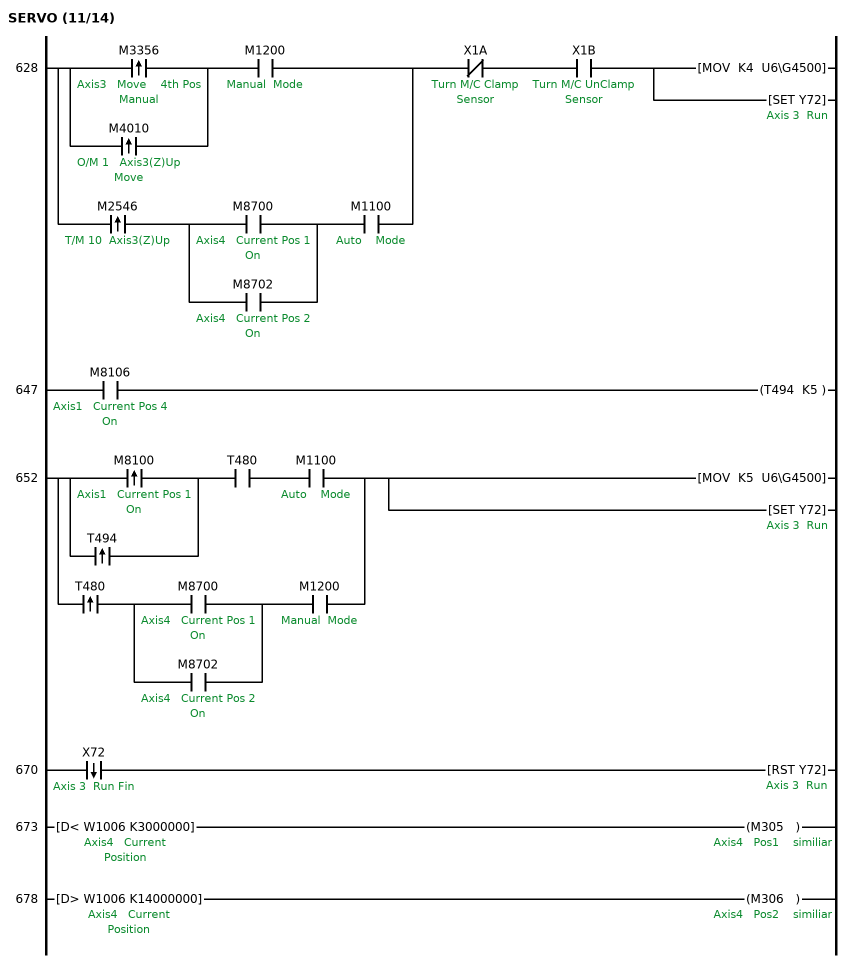
[picture p48: ladder of SERVO, rungs at steps 628 to 678]
628   LDP     M3356  ; Axis3   Move    4th Pos Manual
      ORP     M4010  ; O/M 1   Axis3(Z)Up Move
      AND     M1200  ; Manual  Mode
      LDP     M2546  ; T/M 10  Axis3(Z)Up
      LD      M8700  ; Axis4   Current Pos 1 On
      OR      M8702  ; Axis4   Current Pos 2 On
      ANB
      AND     M1100  ; Auto    Mode
      ORB
      ANI     X1A  ; Turn M/C Clamp Sensor
      AND     X1B  ; Turn M/C UnClamp Sensor
      MOV     K4 U6\G4500
      SET     Y72  ; Axis 3  Run
647   LD      M8106  ; Axis1   Current Pos 4 On
      OUT     T494 K5
652   LDP     M8100  ; Axis1   Current Pos 1 On
      ORP     T494
      AND     T480
      AND     M1100  ; Auto    Mode
      LDP     T480
      LD      M8700  ; Axis4   Current Pos 1 On
      OR      M8702  ; Axis4   Current Pos 2 On
      ANB
      AND     M1200  ; Manual  Mode
      ORB
      MOV     K5 U6\G4500
      SET     Y72  ; Axis 3  Run
670   LDF     X72  ; Axis 3  Run Fin
      RST     Y72  ; Axis 3  Run
673   LDD<    W1006 K3000000  ; Axis4   Current Position
      OUT     M305  ; Axis4   Pos1    similiar
678   LDD>    W1006 K14000000  ; Axis4   Current Position
      OUT     M306  ; Axis4   Pos2    similiar
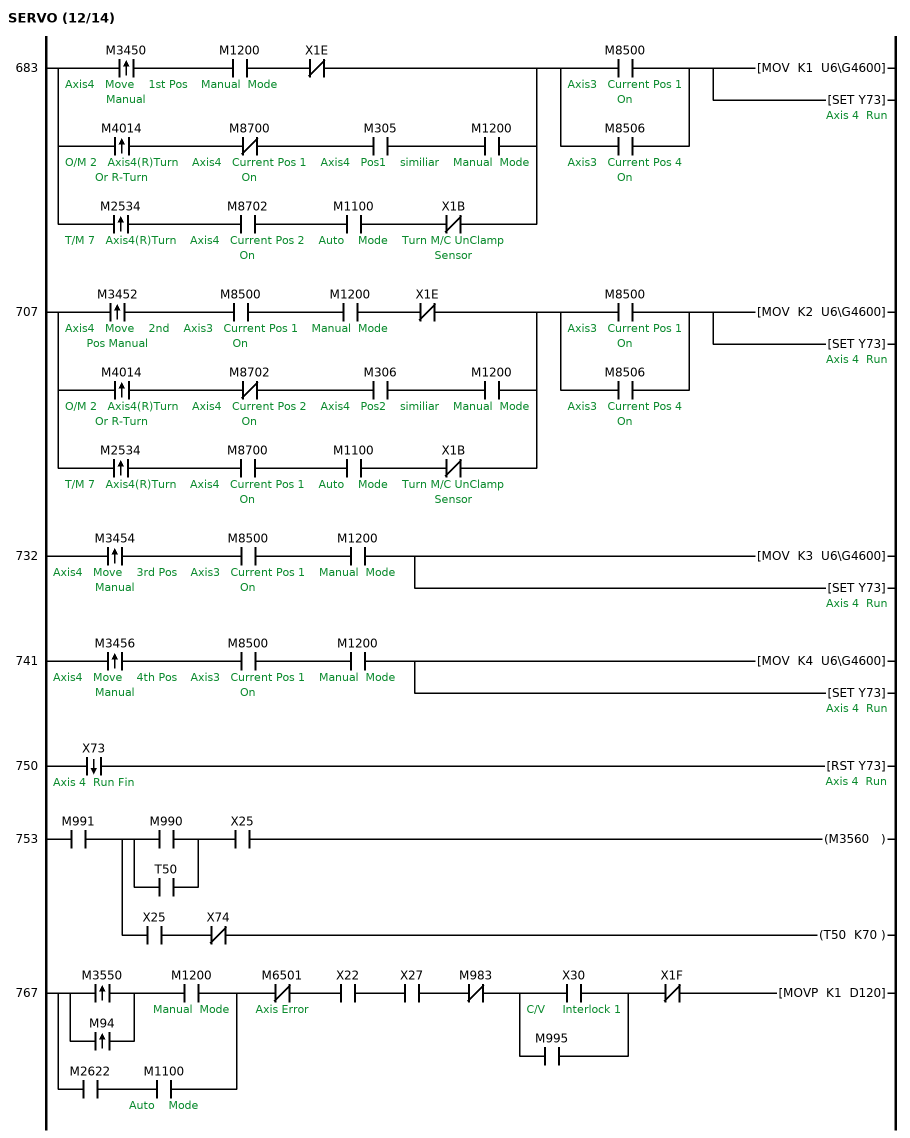
683   LDP     M3450  ; Axis4   Move    1st Pos Manual
      AND     M1200  ; Manual  Mode
      ANI     X1E
      LDP     M4014  ; O/M 2   Axis4(R)Turn Or R-Turn
      ANI     M8700  ; Axis4   Current Pos 1 On
      AND     M305  ; Axis4   Pos1    similiar
      AND     M1200  ; Manual  Mode
      ORB
      LDP     M2534  ; T/M 7   Axis4(R)Turn
      AND     M8702  ; Axis4   Current Pos 2 On
      AND     M1100  ; Auto    Mode
      ANI     X1B  ; Turn M/C UnClamp Sensor
      ORB
      LD      M8500  ; Axis3   Current Pos 1 On
      OR      M8506  ; Axis3   Current Pos 4 On
      ANB
      MOV     K1 U6\G4600
      SET     Y73  ; Axis 4  Run
707   LDP     M3452  ; Axis4   Move    2nd Pos Manual
      AND     M8500  ; Axis3   Current Pos 1 On
      AND     M1200  ; Manual  Mode
      ANI     X1E
      LDP     M4014  ; O/M 2   Axis4(R)Turn Or R-Turn
      ANI     M8702  ; Axis4   Current Pos 2 On
      AND     M306  ; Axis4   Pos2    similiar
      AND     M1200  ; Manual  Mode
      ORB
      LDP     M2534  ; T/M 7   Axis4(R)Turn
      AND     M8700  ; Axis4   Current Pos 1 On
      AND     M1100  ; Auto    Mode
      ANI     X1B  ; Turn M/C UnClamp Sensor
      ORB
      LD      M8500  ; Axis3   Current Pos 1 On
      OR      M8506  ; Axis3   Current Pos 4 On
      ANB
      MOV     K2 U6\G4600
      SET     Y73  ; Axis 4  Run
732   LDP     M3454  ; Axis4   Move    3rd Pos Manual
      AND     M8500  ; Axis3   Current Pos 1 On
      AND     M1200  ; Manual  Mode
      MOV     K3 U6\G4600
      SET     Y73  ; Axis 4  Run
741   LDP     M3456  ; Axis4   Move    4th Pos Manual
      AND     M8500  ; Axis3   Current Pos 1 On
      AND     M1200  ; Manual  Mode
      MOV     K4 U6\G4600
      SET     Y73  ; Axis 4  Run
750   LDF     X73  ; Axis 4  Run Fin
      RST     Y73  ; Axis 4  Run
753   LD      M991
      MPS
      LD      M990
      OR      T50
      ANB
      AND     X25
      OUT     M3560
      MPP
      AND     X25
      ANI     X74
      OUT     T50 K70
767   LDP     M3550
      ORP     M94
      AND     M1200  ; Manual  Mode
      LD      M2622
      AND     M1100  ; Auto    Mode
      ORB
      ANI     M6501  ; Axis Error
      AND     X22
      AND     X27
      ANI     M983
      LD      X30  ; C/V     Interlock 1
      OR      M995
      ANB
      ANI     X1F
      MOVP    K1 D120
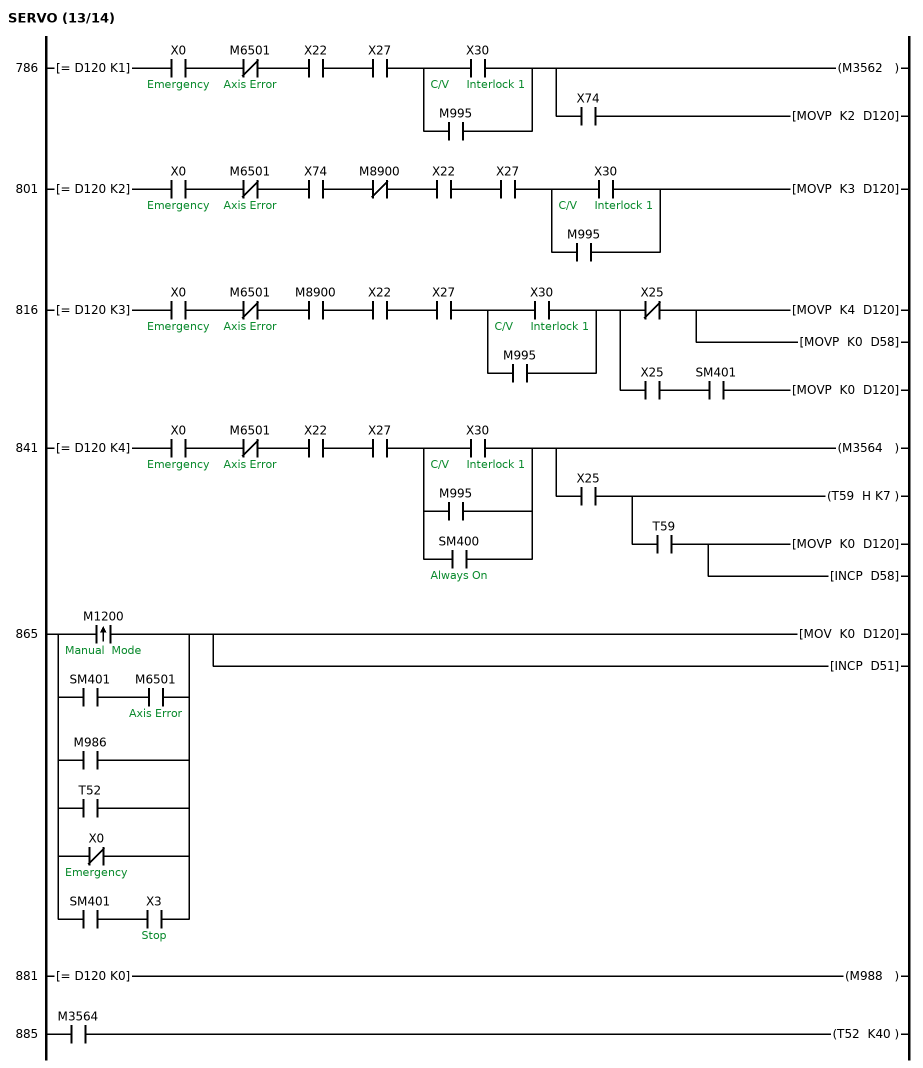
786   LD=     D120 K1
      AND     X0  ; Emergency
      ANI     M6501  ; Axis Error
      AND     X22
      AND     X27
      LD      X30  ; C/V     Interlock 1
      OR      M995
      ANB
      OUT     M3562
      AND     X74
      MOVP    K2 D120
801   LD=     D120 K2
      AND     X0  ; Emergency
      ANI     M6501  ; Axis Error
      AND     X74
      ANI     M8900
      AND     X22
      AND     X27
      LD      X30  ; C/V     Interlock 1
      OR      M995
      ANB
      MOVP    K3 D120
816   LD=     D120 K3
      AND     X0  ; Emergency
      ANI     M6501  ; Axis Error
      AND     M8900
      AND     X22
      AND     X27
      LD      X30  ; C/V     Interlock 1
      OR      M995
      ANB
      MPS
      ANI     X25
      MOVP    K4 D120
      MOVP    K0 D58
      MPP
      AND     X25
      AND     SM401
      MOVP    K0 D120
841   LD=     D120 K4
      AND     X0  ; Emergency
      ANI     M6501  ; Axis Error
      AND     X22
      AND     X27
      LD      X30  ; C/V     Interlock 1
      OR      M995
      OR      SM400  ; Always On
      ANB
      OUT     M3564
      AND     X25
      OUTH    T59 K7
      AND     T59
      MOVP    K0 D120
      INCP    D58
865   LDP     M1200  ; Manual  Mode
      LD      SM401
      AND     M6501  ; Axis Error
      ORB
      OR      M986
      OR      T52
      ORI     X0  ; Emergency
      LD      SM401
      AND     X3  ; Stop
      ORB
      MOV     K0 D120
      INCP    D51
881   LD=     D120 K0
      OUT     M988
885   LD      M3564
      OUT     T52 K40
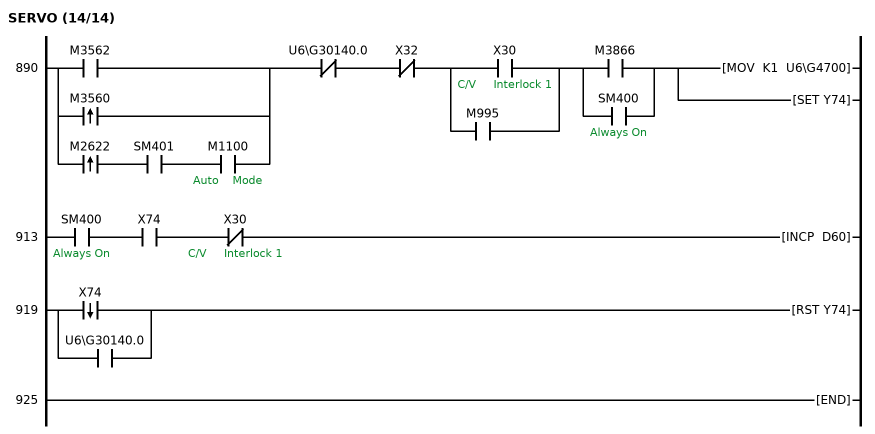
890   LD      M3562
      ORP     M3560
      LDP     M2622
      AND     SM401
      AND     M1100  ; Auto    Mode
      ORB
      ANI     U6\G30140.0
      ANI     X32
      LD      X30  ; C/V     Interlock 1
      OR      M995
      ANB
      LD      M3866
      OR      SM400  ; Always On
      ANB
      MOV     K1 U6\G4700
      SET     Y74
913   LD      SM400  ; Always On
      AND     X74
      ANI     X30  ; C/V     Interlock 1
      INCP    D60
919   LDF     X74
      OR      U6\G30140.0
      RST     Y74
925   END
END_PROGRAM

PROGRAM Y_OUT
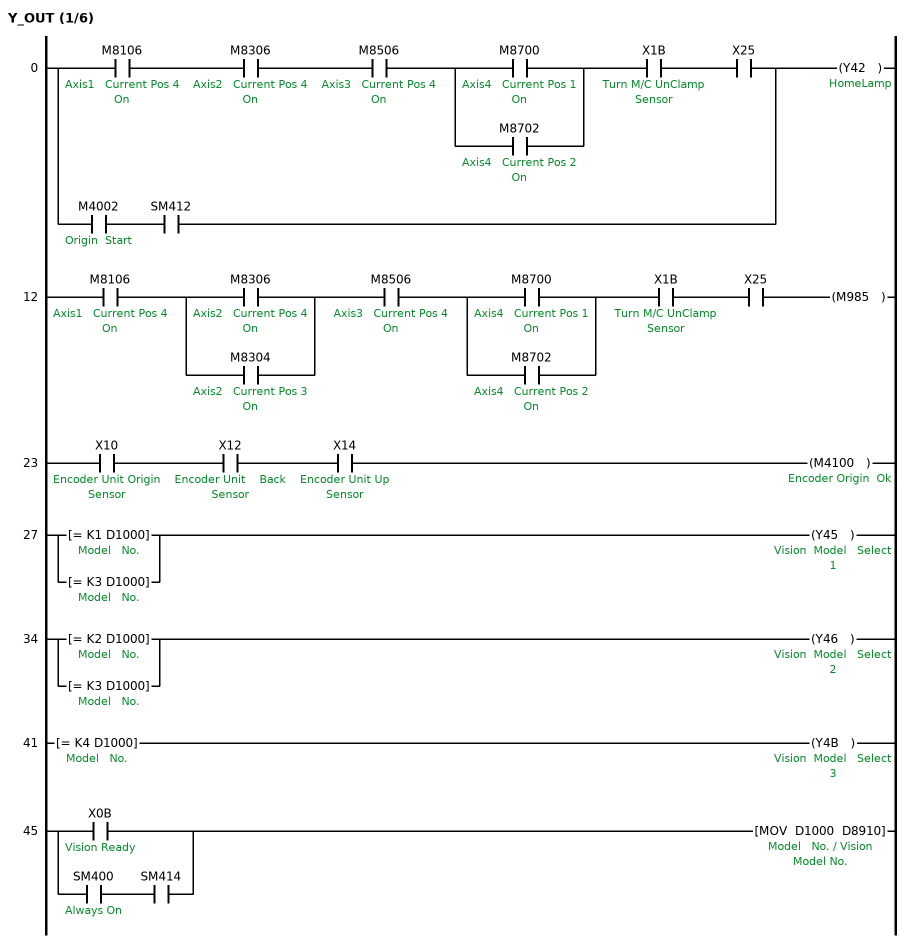
0     LD      M8106  ; Axis1   Current Pos 4 On
      AND     M8306  ; Axis2   Current Pos 4 On
      AND     M8506  ; Axis3   Current Pos 4 On
      LD      M8700  ; Axis4   Current Pos 1 On
      OR      M8702  ; Axis4   Current Pos 2 On
      ANB
      AND     X1B  ; Turn M/C UnClamp Sensor
      AND     X25
      LD      M4002  ; Origin  Start
      AND     SM412
      ORB
      OUT     Y42  ; HomeLamp
12    LD      M8106  ; Axis1   Current Pos 4 On
      LD      M8306  ; Axis2   Current Pos 4 On
      OR      M8304  ; Axis2   Current Pos 3 On
      ANB
      AND     M8506  ; Axis3   Current Pos 4 On
      LD      M8700  ; Axis4   Current Pos 1 On
      OR      M8702  ; Axis4   Current Pos 2 On
      ANB
      AND     X1B  ; Turn M/C UnClamp Sensor
      AND     X25
      OUT     M985
23    LD      X10  ; Encoder Unit Origin Sensor
      AND     X12  ; Encoder Unit    Back    Sensor
      AND     X14  ; Encoder Unit Up Sensor
      OUT     M4100  ; Encoder Origin  Ok
27    LD=     K1 D1000  ; Model   No.
      OR=     K3 D1000  ; Model   No.
      OUT     Y45  ; Vision  Model   Select 1
34    LD=     K2 D1000  ; Model   No.
      OR=     K3 D1000  ; Model   No.
      OUT     Y46  ; Vision  Model   Select 2
41    LD=     K4 D1000  ; Model   No.
      OUT     Y4B  ; Vision  Model   Select 3
45    LD      X0B  ; Vision Ready
      LD      SM400  ; Always On
      AND     SM414
      ORB
      MOV     D1000 D8910  ; Vision Model No.
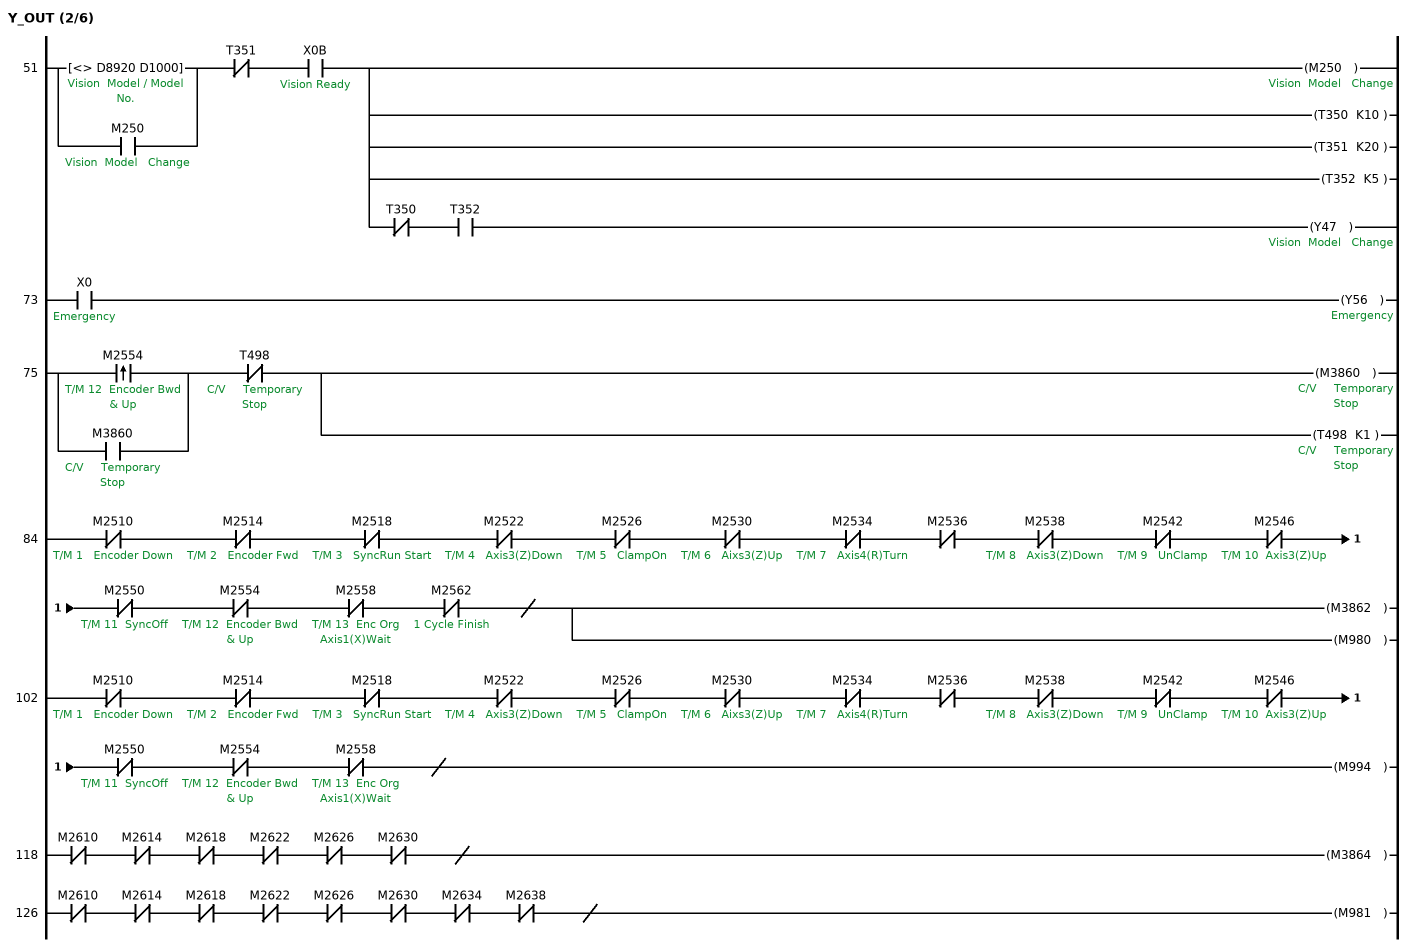
51    LD<>    D8920 D1000  ; Vision  Model / Model   No.
      OR      M250  ; Vision  Model   Change
      ANI     T351
      AND     X0B  ; Vision Ready
      OUT     M250  ; Vision  Model   Change
      OUT     T350 K10
      OUT     T351 K20
      OUT     T352 K5
      ANI     T350
      AND     T352
      OUT     Y47  ; Vision  Model   Change
73    LD      X0  ; Emergency
      OUT     Y56  ; Emergency
75    LDP     M2554  ; T/M 12  Encoder Bwd & Up
      OR      M3860  ; C/V     Temporary  Stop
      ANI     T498  ; C/V     Temporary  Stop
      OUT     M3860  ; C/V     Temporary  Stop
      OUT     T498 K1  ; C/V     Temporary  Stop
84    LDI     M2510  ; T/M 1   Encoder Down
      ANI     M2514  ; T/M 2   Encoder Fwd
      ANI     M2518  ; T/M 3   SyncRun Start
      ANI     M2522  ; T/M 4   Axis3(Z)Down
      ANI     M2526  ; T/M 5   ClampOn
      ANI     M2530  ; T/M 6   Aixs3(Z)Up
      ANI     M2534  ; T/M 7   Axis4(R)Turn
      ANI     M2536
      ANI     M2538  ; T/M 8   Axis3(Z)Down
      ANI     M2542  ; T/M 9   UnClamp
      ANI     M2546  ; T/M 10  Axis3(Z)Up
      ANI     M2550  ; T/M 11  SyncOff
      ANI     M2554  ; T/M 12  Encoder Bwd & Up
      ANI     M2558  ; T/M 13  Enc Org Axis1(X)Wait
      ANI     M2562  ; 1 Cycle Finish
      INV
      OUT     M3862
      OUT     M980
102   LDI     M2510  ; T/M 1   Encoder Down
      ANI     M2514  ; T/M 2   Encoder Fwd
      ANI     M2518  ; T/M 3   SyncRun Start
      ANI     M2522  ; T/M 4   Axis3(Z)Down
      ANI     M2526  ; T/M 5   ClampOn
      ANI     M2530  ; T/M 6   Aixs3(Z)Up
      ANI     M2534  ; T/M 7   Axis4(R)Turn
      ANI     M2536
      ANI     M2538  ; T/M 8   Axis3(Z)Down
      ANI     M2542  ; T/M 9   UnClamp
      ANI     M2546  ; T/M 10  Axis3(Z)Up
      ANI     M2550  ; T/M 11  SyncOff
      ANI     M2554  ; T/M 12  Encoder Bwd & Up
      ANI     M2558  ; T/M 13  Enc Org Axis1(X)Wait
      INV
      OUT     M994
118   LDI     M2610
      ANI     M2614
      ANI     M2618
      ANI     M2622
      ANI     M2626
      ANI     M2630
      INV
      OUT     M3864
126   LDI     M2610
      ANI     M2614
      ANI     M2618
      ANI     M2622
      ANI     M2626
      ANI     M2630
      ANI     M2634
      ANI     M2638
      INV
      OUT     M981
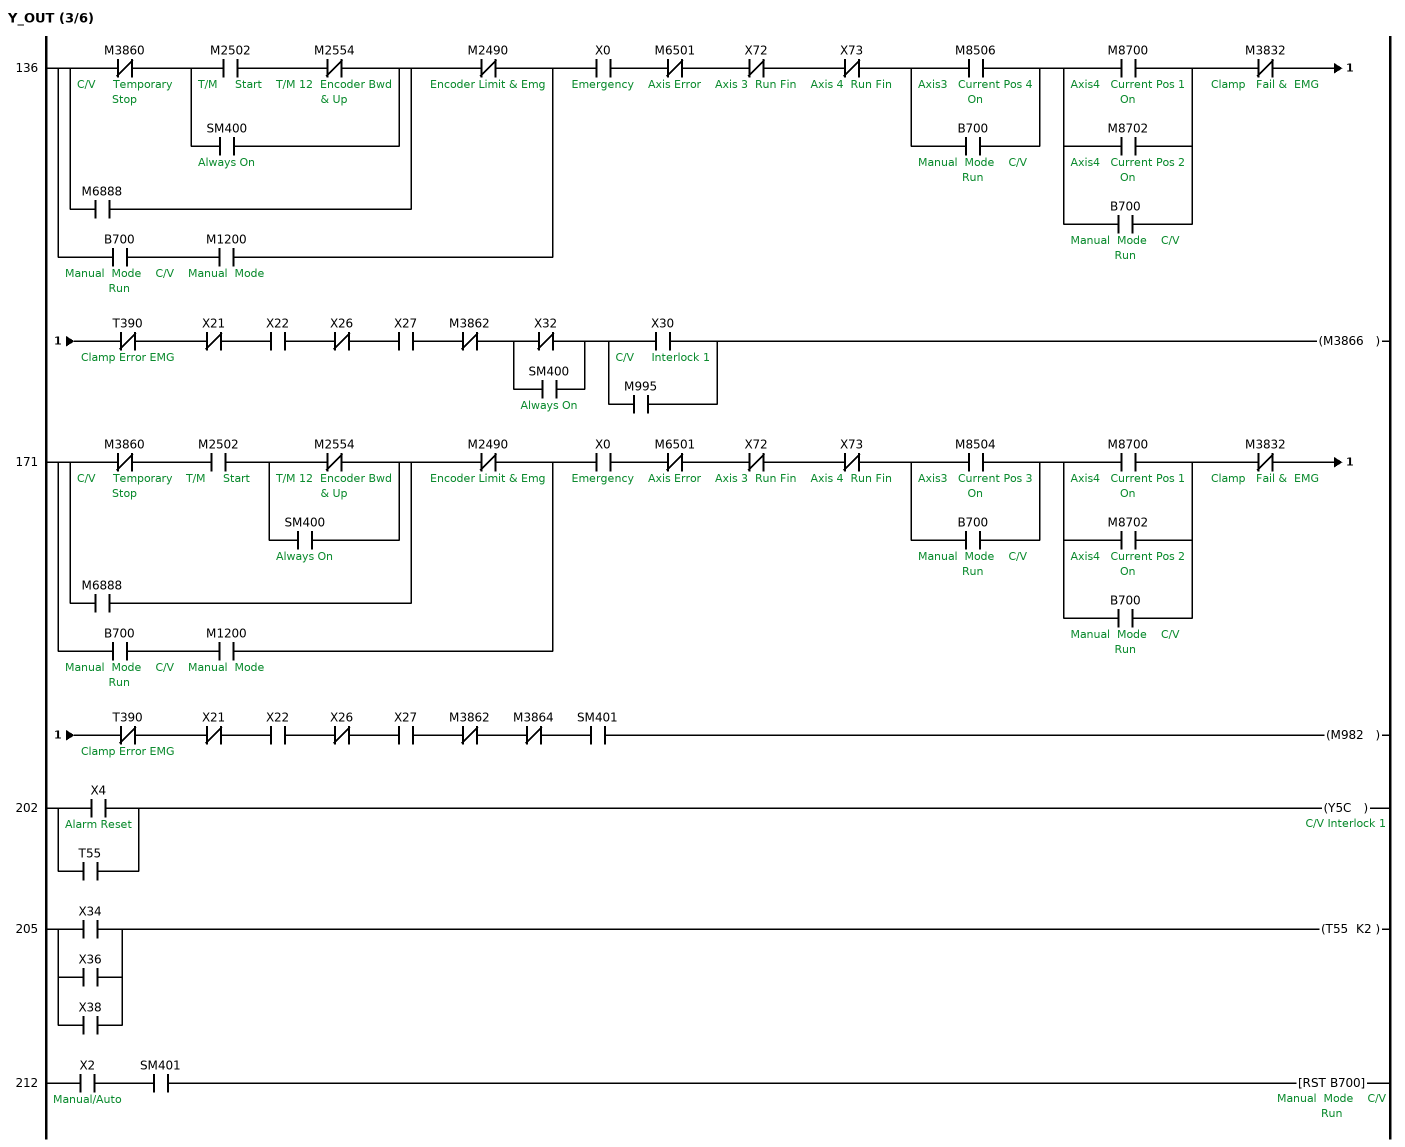
136   LDI     M3860  ; C/V     Temporary  Stop
      LD      M2502  ; T/M     Start
      ANI     M2554  ; T/M 12  Encoder Bwd & Up
      OR      SM400  ; Always On
      ANB
      OR      M6888
      ANI     M2490  ; Encoder Limit & Emg
      LD      B700  ; Manual  Mode    C/V Run
      AND     M1200  ; Manual  Mode
      ORB
      AND     X0  ; Emergency
      ANI     M6501  ; Axis Error
      ANI     X72  ; Axis 3  Run Fin
      ANI     X73  ; Axis 4  Run Fin
      LD      M8506  ; Axis3   Current Pos 4 On
      OR      B700  ; Manual  Mode    C/V Run
      ANB
      LD      M8700  ; Axis4   Current Pos 1 On
      OR      M8702  ; Axis4   Current Pos 2 On
      OR      B700  ; Manual  Mode    C/V Run
      ANB
      ANI     M3832  ; Clamp   Fail &  EMG
      ANI     T390  ; Clamp Error EMG
      ANI     X21
      AND     X22
      ANI     X26
      AND     X27
      ANI     M3862
      LDI     X32
      OR      SM400  ; Always On
      ANB
      LD      X30  ; C/V     Interlock 1
      OR      M995
      ANB
      OUT     M3866
171   LDI     M3860  ; C/V     Temporary  Stop
      AND     M2502  ; T/M     Start
      LDI     M2554  ; T/M 12  Encoder Bwd & Up
      OR      SM400  ; Always On
      ANB
      OR      M6888
      ANI     M2490  ; Encoder Limit & Emg
      LD      B700  ; Manual  Mode    C/V Run
      AND     M1200  ; Manual  Mode
      ORB
      AND     X0  ; Emergency
      ANI     M6501  ; Axis Error
      ANI     X72  ; Axis 3  Run Fin
      ANI     X73  ; Axis 4  Run Fin
      LD      M8504  ; Axis3   Current Pos 3 On
      OR      B700  ; Manual  Mode    C/V Run
      ANB
      LD      M8700  ; Axis4   Current Pos 1 On
      OR      M8702  ; Axis4   Current Pos 2 On
      OR      B700  ; Manual  Mode    C/V Run
      ANB
      ANI     M3832  ; Clamp   Fail &  EMG
      ANI     T390  ; Clamp Error EMG
      ANI     X21
      AND     X22
      ANI     X26
      AND     X27
      ANI     M3862
      ANI     M3864
      AND     SM401
      OUT     M982
202   LD      X4  ; Alarm Reset
      OR      T55
      OUT     Y5C  ; C/V Interlock 1
205   LD      X34
      OR      X36
      OR      X38
      OUT     T55 K2
212   LD      X2  ; Manual/Auto
      AND     SM401
      RST     B700  ; Manual  Mode    C/V Run
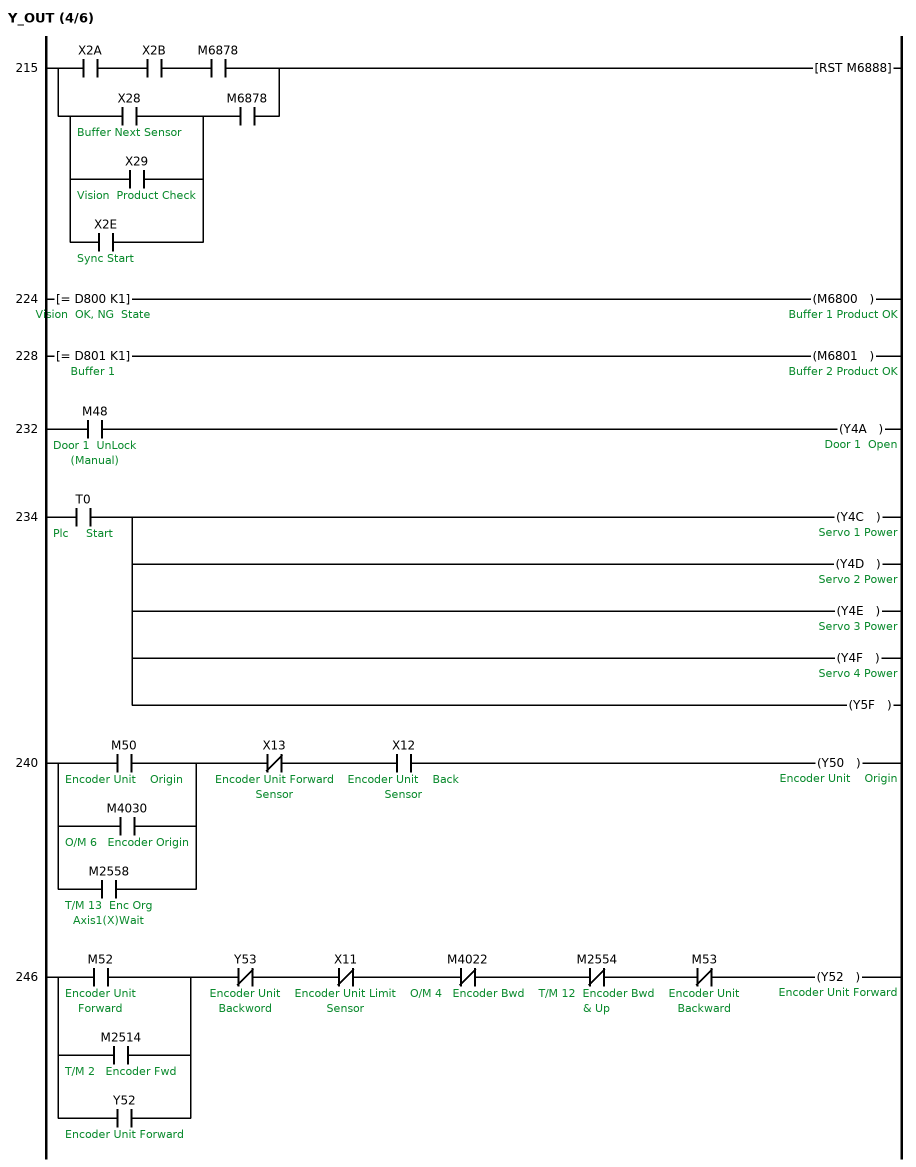
215   LD      X2A
      AND     X2B
      AND     M6878
      LD      X28  ; Buffer Next Sensor
      OR      X29  ; Vision  Product Check
      OR      X2E  ; Sync Start
      AND     M6878
      ORB
      RST     M6888
224   LD=     D800 K1  ; Vision  OK, NG  State
      OUT     M6800  ; Buffer 1 Product OK
228   LD=     D801 K1  ; Buffer 1
      OUT     M6801  ; Buffer 2 Product OK
232   LD      M48  ; Door 1  UnLock  (Manual)
      OUT     Y4A  ; Door 1  Open
234   LD      T0  ; Plc     Start
      OUT     Y4C  ; Servo 1 Power
      OUT     Y4D  ; Servo 2 Power
      OUT     Y4E  ; Servo 3 Power
      OUT     Y4F  ; Servo 4 Power
      OUT     Y5F
240   LD      M50  ; Encoder Unit    Origin
      OR      M4030  ; O/M 6   Encoder Origin
      OR      M2558  ; T/M 13  Enc Org Axis1(X)Wait
      ANI     X13  ; Encoder Unit Forward Sensor
      AND     X12  ; Encoder Unit    Back    Sensor
      OUT     Y50  ; Encoder Unit    Origin
246   LD      M52  ; Encoder Unit    Forward
      OR      M2514  ; T/M 2   Encoder Fwd
      OR      Y52  ; Encoder Unit Forward
      ANI     Y53  ; Encoder Unit Backword
      ANI     X11  ; Encoder Unit Limit Sensor
      ANI     M4022  ; O/M 4   Encoder Bwd
      ANI     M2554  ; T/M 12  Encoder Bwd & Up
      ANI     M53  ; Encoder Unit    Backward
      OUT     Y52  ; Encoder Unit Forward
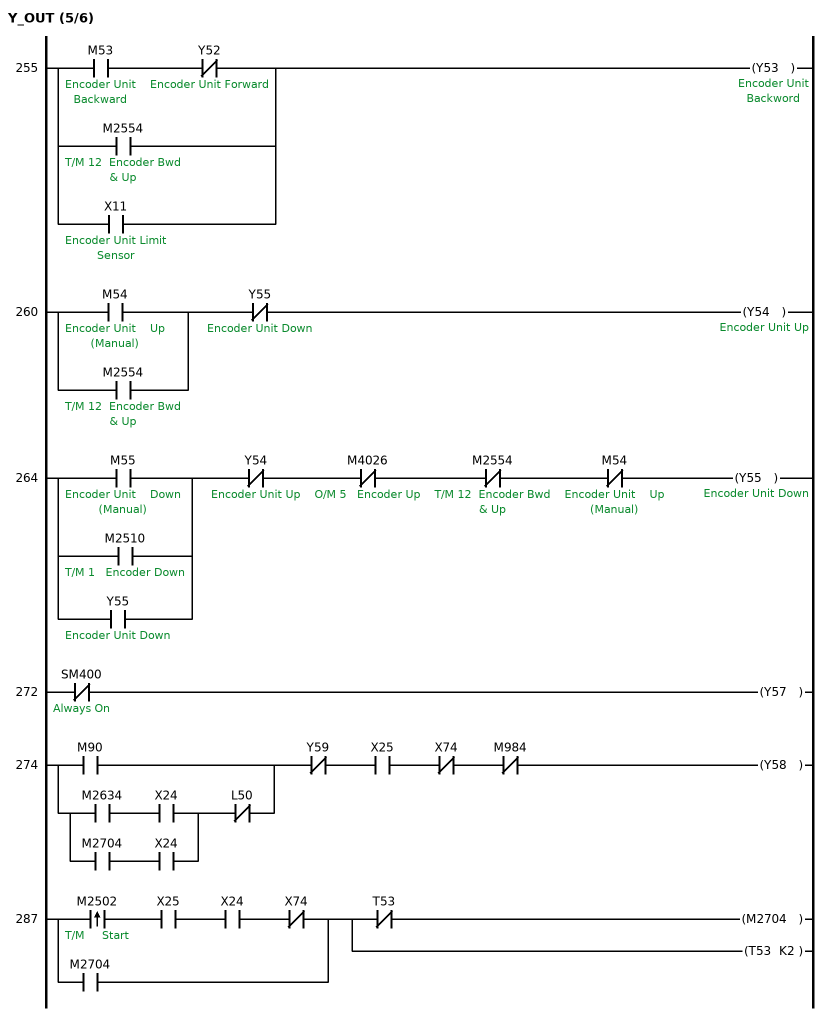
255   LD      M53  ; Encoder Unit    Backward
      ANI     Y52  ; Encoder Unit Forward
      OR      M2554  ; T/M 12  Encoder Bwd & Up
      OR      X11  ; Encoder Unit Limit Sensor
      OUT     Y53  ; Encoder Unit Backword
260   LD      M54  ; Encoder Unit    Up      (Manual)
      OR      M2554  ; T/M 12  Encoder Bwd & Up
      ANI     Y55  ; Encoder Unit Down
      OUT     Y54  ; Encoder Unit Up
264   LD      M55  ; Encoder Unit    Down    (Manual)
      OR      M2510  ; T/M 1   Encoder Down
      OR      Y55  ; Encoder Unit Down
      ANI     Y54  ; Encoder Unit Up
      ANI     M4026  ; O/M 5   Encoder Up
      ANI     M2554  ; T/M 12  Encoder Bwd & Up
      ANI     M54  ; Encoder Unit    Up      (Manual)
      OUT     Y55  ; Encoder Unit Down
272   LDI     SM400  ; Always On
      OUT     Y57
274   LD      M90
      LD      M2634
      AND     X24
      LD      M2704
      AND     X24
      ORB
      ANI     L50
      ORB
      ANI     Y59
      AND     X25
      ANI     X74
      ANI     M984
      OUT     Y58
287   LDP     M2502  ; T/M     Start
      AND     X25
      AND     X24
      ANI     X74
      OR      M2704
      MPS
      ANI     T53
      OUT     M2704
      MPP
      OUT     T53 K2
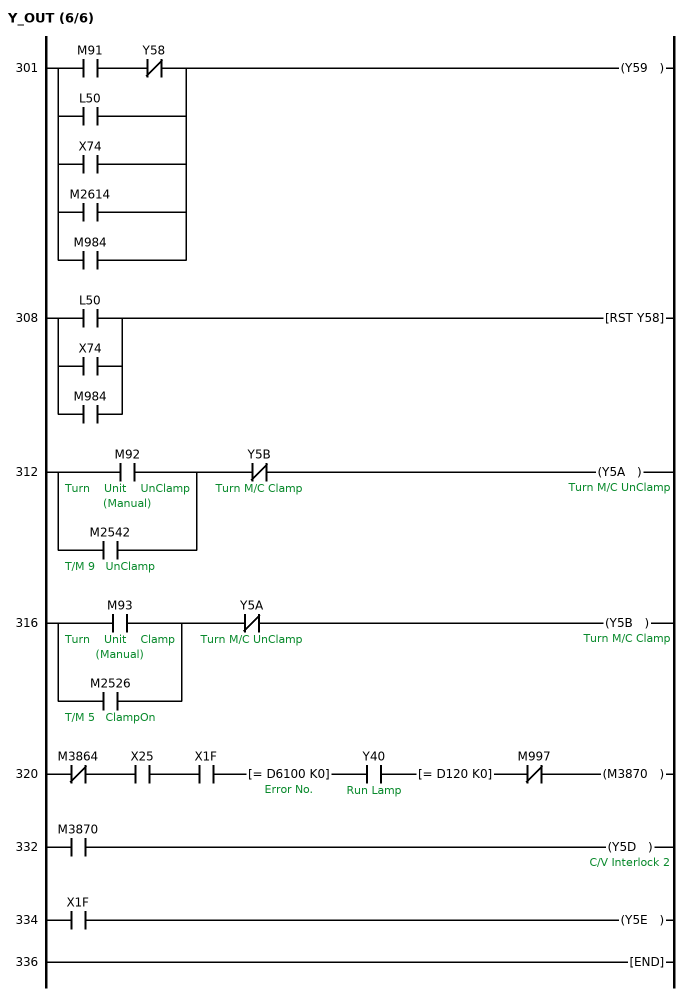
301   LD      M91
      ANI     Y58
      OR      L50
      OR      X74
      OR      M2614
      OR      M984
      OUT     Y59
308   LD      L50
      OR      X74
      OR      M984
      RST     Y58
312   LD      M92  ; Turn    Unit    UnClamp (Manual)
      OR      M2542  ; T/M 9   UnClamp
      ANI     Y5B  ; Turn M/C Clamp
      OUT     Y5A  ; Turn M/C UnClamp
316   LD      M93  ; Turn    Unit    Clamp   (Manual)
      OR      M2526  ; T/M 5   ClampOn
      ANI     Y5A  ; Turn M/C UnClamp
      OUT     Y5B  ; Turn M/C Clamp
320   LDI     M3864
      AND     X25
      AND     X1F
      AND=    D6100 K0  ; Error No.
      AND     Y40  ; Run Lamp
      AND=    D120 K0
      ANI     M997
      OUT     M3870
332   LD      M3870
      OUT     Y5D  ; C/V Interlock 2
334   LD      X1F
      OUT     Y5E
336   END
END_PROGRAM

PROGRAM PB
0     END
END_PROGRAM

// device comments not shown above
X0A  ; Vision Trigger On ark
X2C  ; Transfer Jig    Check 1
X2D  ; Transfer Jig    Check 2
X2F  ; Transfer Product Check 1
X68  ; Axis 1  Error
X69  ; Axis 2  Error
X6A  ; Axis 3  Error
X6B  ; Axis 4  Error
X6C  ; Axis 1  Busy
X6D  ; Axis 2  Busy
X6E  ; Axis 3  Busy
X6F  ; Axis 4  Busy
X200  ; PunchingFWD-1   Px
X201  ; PunchingREV-1   Px
X202  ; PunchingFWD-2   Px
X203  ; PunchingREV-2   Px
X204  ; PunchingFWD-3   Px
X205  ; PunchingREV-3   Px
X206  ; PunchingCHECK   P/H
X207  ; PunchingUnCLAMP Px
X208  ; Burring FWD-1   Px
X209  ; Burring REV-1   Px
X20A  ; Burring FWD-2   Px
X20B  ; Burring REV-2   Px
X20C  ; Burring FWD-3   Px
X20D  ; Burring REV-3   Px
X20E  ; Burring CHECK   P/H
X20F  ; Burring UnCLAMP  Px
X210  ; 펀칭 양수 1
X211  ; 버링 양수 1
X212  ; 펀칭 양수 2
X213  ; 버링 양수 2
X214  ; PunchingCLAMP   Px
X215  ; Burring CLAMP    Px
X216  ; Spider  Check
X217  ; 유압체크
X21C  ; 펀칭 비상정지
X21D  ; 퍼칭 리셋
X21E  ; 버링 비상정지
X21F  ; 버링 리셋
Y64  ; Axis 1  Stop
Y65  ; Axis 2  Stop
Y66  ; Axis 3  Stop
Y67  ; Axis 4  Stop
Y68  ; Axis 1  Jog+
Y69  ; Axis 1  Jog-
Y6A  ; Axis 2  Jog+
Y6B  ; Axis 2  Jog-
Y6C  ; Axis 3  Jog+
Y6D  ; Axis 3  Jog-
Y6E  ; Axis 4  Jog+
Y6F  ; Axis 4  Jog-
Y224  ; PunchingFWD-1
Y225  ; PunchingREV-1
Y226  ; PunchingFWD-2
Y227  ; PunchingREV-2
Y228  ; PunchingFWD-3
Y229  ; PunchingREV-3
Y22A  ; Burring FWD-1
Y22B  ; Burring REV-1
Y22C  ; Burring FWD-2
Y22D  ; Burring REV-2
Y22E  ; Burring FWD-3
Y22F  ; Burring REV-3
Y23A  ; PunchingCLAMP
Y23B  ; PunchingUnCLAMP
Y23C  ; Burring CLAMP
Y23D  ; Burring UnCLAMP
M20  ; Manual/ Auto    Select
M1701  ; Model   No.1
M1702  ; Model   No.2
M1703  ; Model   No.3
M1704  ; Model   No.4
M1705  ; Model   No.5
M1706  ; Model   No.6
M1707  ; Model   No.7
M1708  ; Model   No.8
M1709  ; Model   No.9
M1710  ; Model   No.10
M2010  ; A/M 1   Wait    Vision  Product
M3820  ; Vision  Check & delay
M6022  ; Tact    Time    Restart 2
T210  ; A/M 1   Wait    Vision  Product
T395  ; Y이동
T432  ; Encoder Unit    Origin  OffDelay
T800  ; Vision  Check & delay
T902  ; 펀칭 양수 딜레이 1
T904  ; 펀칭 Clamp On
T906  ; 펀칭 시작
T908  ; 펀칭 완료 후 펀칭 후진
T910  ; 펀칭후진 완료 후 Clamp 후진
T912  ; 펀칭완료
T952  ; 버링 양수 딜레이 1
T954  ; 버링 Clamp On
T956  ; 버링 시작
T958  ; 버링완료 후 버링 후진
T960  ; 버링후진 완료 후 Clamp 후진
T962  ; 버링완료
